FUNCTION_BLOCK Test_TimeAsString_ms EXTENDS TUnitTestBase
VAR
END_VAR

METHOD  Execute
VAR_INST
    TimeStruct : TIMESTRUCT := (wHour := 6, wMinute := 5, wSecond := 4, wMilliseconds := 135);
END_VAR
Assertion.AssertEquals_STRING(
    Expected := '06:05:04.135',
    Actual   := F_TimeAsString_ms(TimeStruct),
    ObjectName := _TestName,
    VariableName  := 'F_TimeAsString_ms(TimeStruct)');


Test_Finished();
END_METHOD

END_FUNCTION_BLOCK

(* stored: Version 1.1.0.1, ProductVersion 3.1.4024.3
   POU Test_TimeAsString_ms: Id {cfe81a32-3eca-0666-0352-ea68d5a05067}, SpecialFunc None
   Method Execute: Id {91043b95-58a1-0ea0-2630-f27f3dd72dd2} *)
